# EPICS substitutions: hugo/source/examples/test/el6022/ecmcEL6022_string.substitutions
file "ecmcEcSlave.template"
{
  pattern {}
          {}
}

file "ecmcEL6022-chX_string.template"
{
  pattern {CH_ID, PLC_ID, NELM }
          {01,    0,      22   }
          {02,    1,      22   }
}
